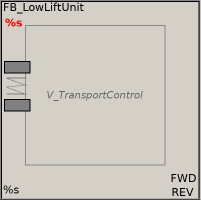
VISUALIZATION V_LowLiftUnit  // 201x200
VAR_IN_OUT
	{attribute 'VAR_IN_OUT_AS_POINTER'}
	fbFunction		: FB_LowLiftUnit;	
END_VAR
    Rectangle (0,0 200x200), colour toggle: fbFunction.BaseFunctionData.ZoneOrders[1].Drive_Run OR fbFunction.BaseFunctionData.ZoneOrders[1].Drive_RunRev
    Rectangle (0,180 200x20), "%s", text variable: fbFunction.ConfigFunction.FunctionName
    Label (0,0 200x15), "FB_LowLiftUnit"
    Label (166,172 35x13), "FWD", invisible if: NOT fbFunction.BaseFunctionData.ZoneOrders[1].Drive_Run
    Label (165,185 35x15), "REV", invisible if: NOT fbFunction.BaseFunctionData.ZoneOrders[1].Drive_RunRev
    Frame (25,25 140x140)
        shows V_TransportControl(TransportControl := fbFunction.fbTransportControl, ZoneData := fbFunction.ZoneData[1])
    Polyline (26,78) (7,78) (26,85) (7,87) (26,94) (7,94), colour toggle: fbFunction.HW_Outputs.Drive_Run_Up OR fbFunction.HW_Outputs.Drive_Run_Down
    Rectangle (4,99 26x12), tooltip "Lower lift sensor", colour toggle: fbFunction.HW_Inputs.Sensor_Pos_Down
    Rectangle (4,61 26x12), tooltip "Upper lift sensor", colour toggle: fbFunction.HW_Inputs.Sensor_Pos_Up
    Rectangle (2,15 194x16), "%s", tooltip "%s", text variable: fbFunction.FunctionData.ErrorData.Error.ErrorCode.Conv, invisible if: fbFunction.FunctionData.ErrorData.ErrorState = E_ErrorState.OPERATIONAL
        p4168582468: fbFunction.FunctionData.ErrorData.Error.ErrorParam
END_VISUALIZATION

(* stored: Version 1.1.0.1, ProductVersion 3.1.4024.9
   Visu V_LowLiftUnit: Id {5b7065e4-5162-4a3f-a66d-11ddcddc0a77} *)
